// TIA Portal V18 export
DATA_BLOCK "SS1_CPU1215_AO_Vars"   // DB11012
{ S7_Optimized_Access := 'FALSE' }
VERSION : 0.1
// stored: AutoNumber false, DBAccessibleFromOPCUA true, IsOnlyStoredInLoadMemory false, IsWriteProtectedInAS false
   VAR
      AO1 { S7_SetPoint := 'True'} : "UDT_AOadv";
      AO2 { S7_SetPoint := 'True'} : "UDT_AOadv";
   END_VAR
BEGIN
   AO1.rInput := 0.0;
   AO1.cMOA := 16#01;
   AO1.cFuncSystemID := 1;
   AO1.cFuncVar := 1;
   AO1.cMemory := 16#00;
   AO1.rManOutput := 60.0;
   AO1.iOutput := 11060;
   AO2.rInput := 0.0;
   AO2.cMOA := 16#00;
   AO2.cFuncSystemID := 16#00;
   AO2.cFuncVar := 16#00;
   AO2.cMemory := 16#00;
   AO2.rManOutput := 0.0;
   AO2.iOutput := 0;
END_DATA_BLOCK
